{attribute addProperty BoxType "KL1501"}
{attribute addProperty Id "Channel_1Channel_C961C78600"}
{attribute addProperty CRC "3532189323"}
{attribute addProperty SizeInBites "0"}
{attribute addProperty SizeInBytes "0"}
TYPE KL1501_D288EE8B :
STRUCT
	{attribute addProperty Name "Channel_1"}
	Channel_1 : Channel_C961C786;
END_STRUCT
END_TYPE

(* stored: Version 1.2.0.0, ProductVersion 3.1.4024.9
   DUT KL1501_D288EE8B: Id {4cb7d83c-ab12-4006-bfdf-96c371d31fd3} *)
